PROGRAM MAIN
VAR
END_VAR

END_PROGRAM

(* stored: Version 1.1.0.1
   POU MAIN: Id {204bbc62-1769-42bb-8b48-0dfa2fe581ab} *)
